(* Logix 5000 project; controller RG_Chopper vendor 1 type 14 code 235 rev 32.12; software revision 32.04; part 2 of 6 *)

ADD_ON_INSTRUCTION PUSH_PUSH_PB   (* revision 1.0, vendor JBT Food Tech *)
// Push Push (Dual State) Push Button
// Push - On; Push - Off
// Revision note:
// Rev 1.0 - 9/8/2010 - KM
VAR_INPUT
   HMI_PB : BOOL; {required}
   One_Shot : BOOL;
END_VAR
VAR_OUTPUT
   S_Out : BOOL; {access Read Only}
END_VAR
VAR_INPUT
   L_Out : BOOL; {visible}
END_VAR

ROUTINE Logic   (* ladder *)
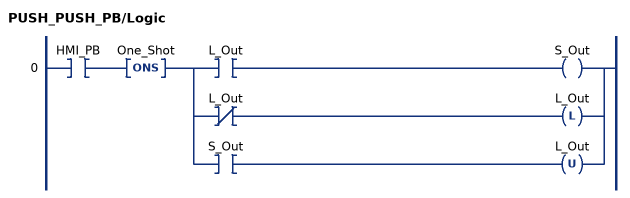
   0: XIC(HMI_PB)ONS(One_Shot)[XIC(L_Out) OTE(S_Out) ,XIO(L_Out) OTL(L_Out) ,XIC(S_Out) OTU(L_Out) ];
END_ROUTINE
END_ADD_ON_INSTRUCTION

ADD_ON_INSTRUCTION TD_TA_TP_4PORT_IOL   (* revision 1.0, vendor ifm efector *)
// Cyclic Data with Diagnostics
// Revision note:
// 4/27/17
VAR_IN_OUT
   PLC_Input : INT[123]; {required}
END_VAR
VAR_INPUT
   Port_Process_Data_Size : INT := 4; {visible}
   Port_Number : INT; {visible}
   Temp_Value_Gradient : REAL := 0.1; {visible}
END_VAR
VAR_OUTPUT
   Temperature : REAL; {access Read Only, visible}
   Vendor_ID : INT; {access Read Only, visible}
   Device_ID : INT; {access Read Only, visible}
   Datastorage_Error : BOOL; {access Read Only, visible}
   Process_Data : INT; {access Read Only}
   Device_Not_Connected : BOOL; {access Read Only, visible}
   IOL_Mode : BOOL; {access Read Only, visible}
   Invalid_Data : BOOL; {access Read Only, visible}
   Wrong_VID_DID : BOOL; {access Read Only, visible}
END_VAR
VAR
   RealPort_Num : INT; {access None}
   Offset_Address : INT; {access None}
   Process_PDI : INT; {access None}
   Process_Offset : INT; {access None}
   Offset_StatusFlgs : INT; {access None}
   StatusFlgs_Offset : INT; {access None}
   Data_Size : INT; {access None}
END_VAR

ROUTINE Logic   (* ladder *)
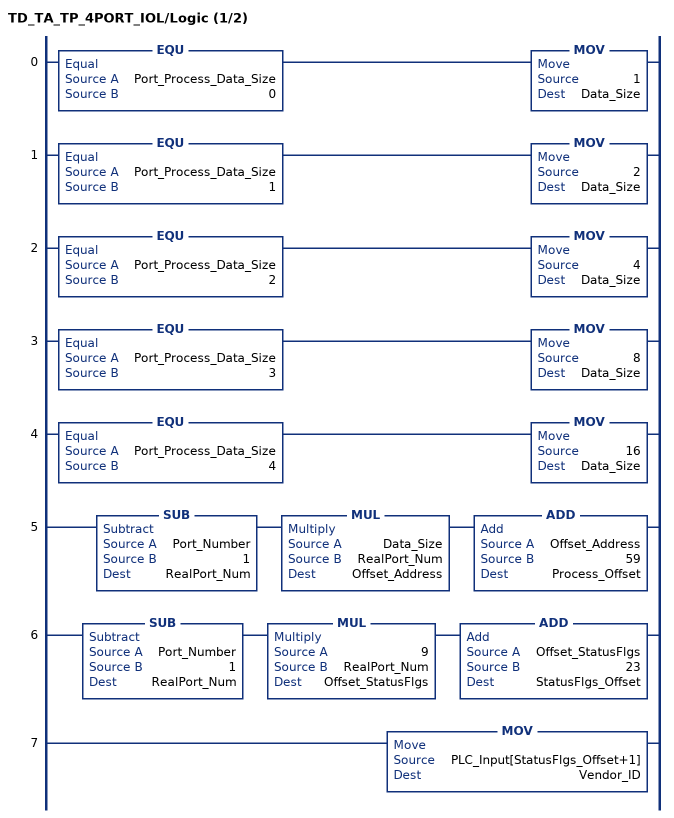
   0: EQU(Port_Process_Data_Size,0)MOV(1,Data_Size);
   1: EQU(Port_Process_Data_Size,1)MOV(2,Data_Size);
   2: EQU(Port_Process_Data_Size,2)MOV(4,Data_Size);
   3: EQU(Port_Process_Data_Size,3)MOV(8,Data_Size);
   4: EQU(Port_Process_Data_Size,4)MOV(16,Data_Size);
   5: SUB(Port_Number,1,RealPort_Num)MUL(Data_Size,RealPort_Num,Offset_Address)ADD(Offset_Address,59,Process_Offset);
   6: SUB(Port_Number,1,RealPort_Num)MUL(9,RealPort_Num,Offset_StatusFlgs)ADD(Offset_StatusFlgs,23,StatusFlgs_Offset);
   7: MOV(PLC_Input[StatusFlgs_Offset+1],Vendor_ID);
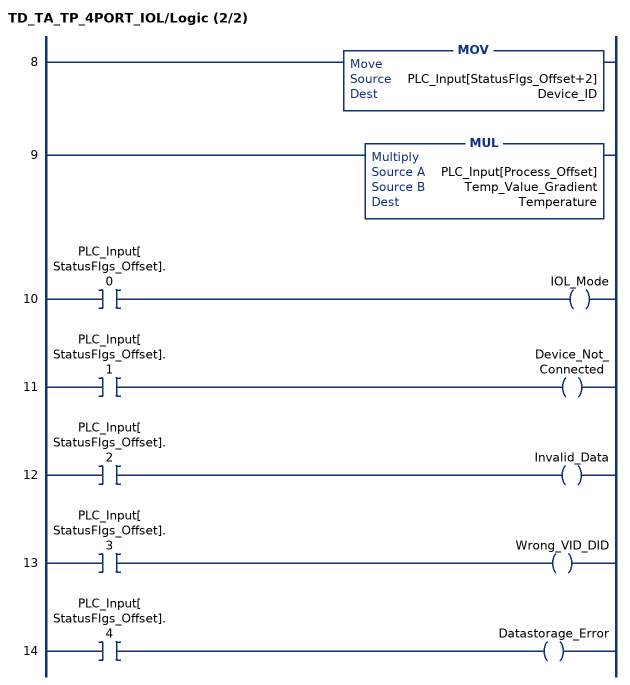
   8: MOV(PLC_Input[StatusFlgs_Offset+2],Device_ID);
   9: MUL(PLC_Input[Process_Offset],Temp_Value_Gradient,Temperature);
   10: XIC(PLC_Input[StatusFlgs_Offset].0)OTE(IOL_Mode);
   11: XIC(PLC_Input[StatusFlgs_Offset].1)OTE(Device_Not_Connected);
   12: XIC(PLC_Input[StatusFlgs_Offset].2)OTE(Invalid_Data);
   13: XIC(PLC_Input[StatusFlgs_Offset].3)OTE(Wrong_VID_DID);
   14: XIC(PLC_Input[StatusFlgs_Offset].4)OTE(Datastorage_Error);
END_ROUTINE
END_ADD_ON_INSTRUCTION

ADD_ON_INSTRUCTION TD_TA_TP_8PORT_IOL   (* revision 1.0, vendor ifm efector *)
// Cyclic Data with Diagnostics
// Revision note:
// 4/27/17
VAR_IN_OUT
   PLC_Input : INT[223]; {required}
END_VAR
VAR_INPUT
   Port_Process_Data_Size : INT := 4; {visible}
   Port_Number : INT; {visible}
   Temp_Value_Gradient : REAL := 0.1; {visible}
END_VAR
VAR_OUTPUT
   Temperature : REAL; {access Read Only, visible}
   Vendor_ID : INT; {access Read Only, visible}
   Device_ID : INT; {access Read Only, visible}
   Datastorage_Error : BOOL; {access Read Only, visible}
   Process_Data : INT; {access Read Only}
   Device_Not_Connected : BOOL; {access Read Only, visible}
   IOL_Mode : BOOL; {access Read Only, visible}
   Invalid_Data : BOOL; {access Read Only, visible}
   Wrong_VID_DID : BOOL; {access Read Only, visible}
END_VAR
VAR
   RealPort_Num : INT; {access None}
   Offset_Address : INT; {access None}
   Process_PDI : INT; {access None}
   Process_Offset : INT; {access None}
   Offset_StatusFlgs : INT; {access None}
   StatusFlgs_Offset : INT; {access None}
   Data_Size : INT; {access None}
END_VAR

ROUTINE Logic   (* ladder *)
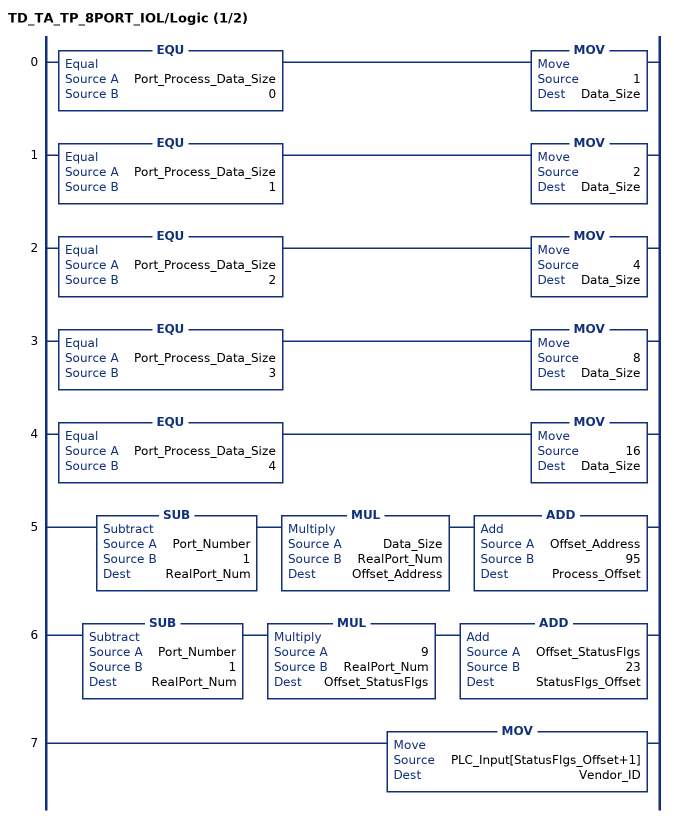
   0: EQU(Port_Process_Data_Size,0)MOV(1,Data_Size);
   1: EQU(Port_Process_Data_Size,1)MOV(2,Data_Size);
   2: EQU(Port_Process_Data_Size,2)MOV(4,Data_Size);
   3: EQU(Port_Process_Data_Size,3)MOV(8,Data_Size);
   4: EQU(Port_Process_Data_Size,4)MOV(16,Data_Size);
   5: SUB(Port_Number,1,RealPort_Num)MUL(Data_Size,RealPort_Num,Offset_Address)ADD(Offset_Address,95,Process_Offset);
   6: SUB(Port_Number,1,RealPort_Num)MUL(9,RealPort_Num,Offset_StatusFlgs)ADD(Offset_StatusFlgs,23,StatusFlgs_Offset);
   7: MOV(PLC_Input[StatusFlgs_Offset+1],Vendor_ID);
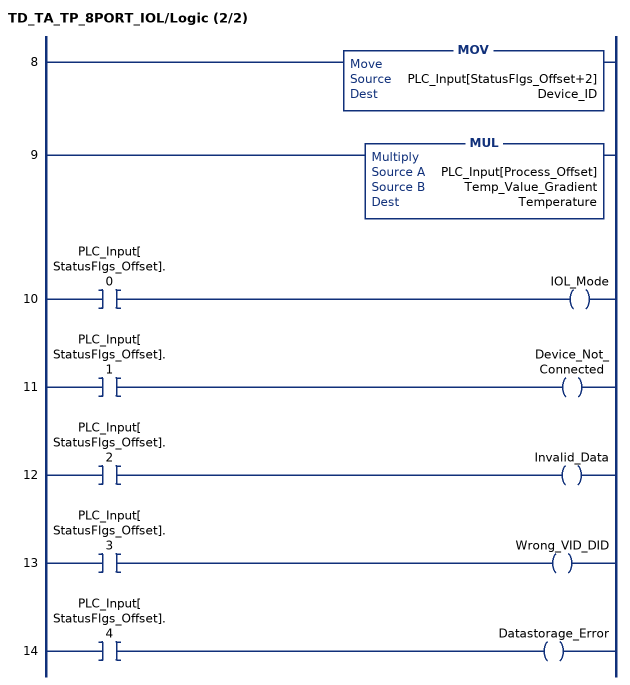
   8: MOV(PLC_Input[StatusFlgs_Offset+2],Device_ID);
   9: MUL(PLC_Input[Process_Offset],Temp_Value_Gradient,Temperature);
   10: XIC(PLC_Input[StatusFlgs_Offset].0)OTE(IOL_Mode);
   11: XIC(PLC_Input[StatusFlgs_Offset].1)OTE(Device_Not_Connected);
   12: XIC(PLC_Input[StatusFlgs_Offset].2)OTE(Invalid_Data);
   13: XIC(PLC_Input[StatusFlgs_Offset].3)OTE(Wrong_VID_DID);
   14: XIC(PLC_Input[StatusFlgs_Offset].4)OTE(Datastorage_Error);
END_ROUTINE
END_ADD_ON_INSTRUCTION

ADD_ON_INSTRUCTION TD_TA_TP_AL1020_IOL   (* revision 1.4, vendor ifm efector *)
// Cyclic Data with Diagnostics
// Revision note:
// Supports TDxxxx, TA2xxx, TP3xxx, TP9xxx
VAR_INPUT
   Port_Number : INT; {visible}
END_VAR
VAR_IN_OUT
   ioarybPLC_Input : INT[194]; {required}
END_VAR
VAR_OUTPUT
   Temp_Value : REAL; {access Read Only, required}
END_VAR
VAR_INPUT
   Temp_Value_Gradient : REAL := 0.1; {visible}
END_VAR
VAR_OUTPUT
   Vendor_ID : INT; {access Read Only, required}
   Device_ID : INT; {access Read Only, required}
   IOLinkmode_active : BOOL; {access Read Only, required}
   IOLink_communication : BOOL; {access Read Only, required}
   Device_Connected : BOOL; {access Read Only, required}
   Valid_Process_Data : BOOL; {access Read Only, required}
   Datastorage_error : BOOL; {access Read Only, required}
END_VAR
VAR
   ARYbInternInputData : INT[26]; {access None}
   Port1 : BOOL; {access None}
   Port2 : BOOL; {access None}
   Port3 : BOOL; {access None}
   Port4 : BOOL; {access None}
   Port5 : BOOL; {access None}
   Port6 : BOOL; {access None}
   Port7 : BOOL; {access None}
   Port8 : BOOL; {access None}
   Process_SWPB : INT; {access None}
END_VAR

ROUTINE Logic   (* ladder *)
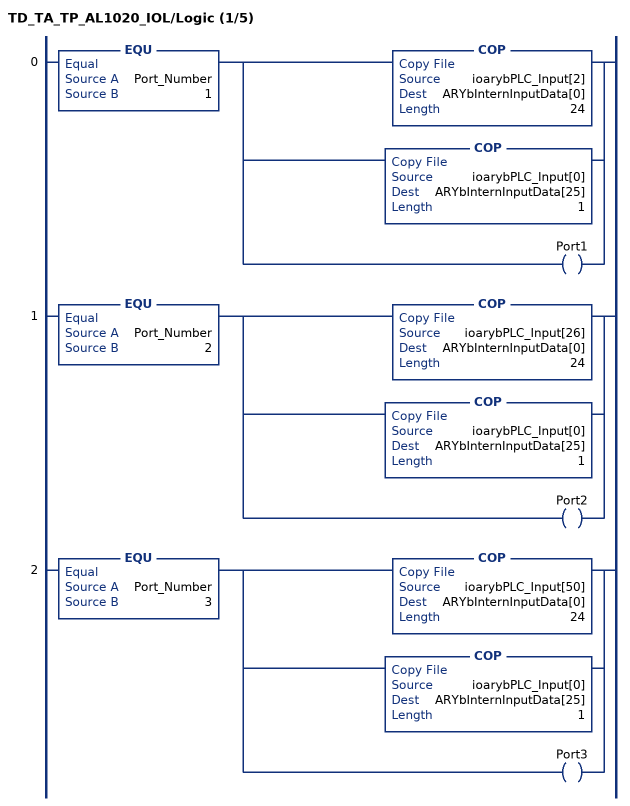
   0: EQU(Port_Number,1)[COP(ioarybPLC_Input[2],ARYbInternInputData[0],24) ,[COP(ioarybPLC_Input[0],ARYbInternInputData[25],1) ,OTE(Port1) ] ];
   1: EQU(Port_Number,2)[COP(ioarybPLC_Input[26],ARYbInternInputData[0],24) ,[COP(ioarybPLC_Input[0],ARYbInternInputData[25],1) ,OTE(Port2) ] ];
   2: EQU(Port_Number,3)[COP(ioarybPLC_Input[50],ARYbInternInputData[0],24) ,[COP(ioarybPLC_Input[0],ARYbInternInputData[25],1) ,OTE(Port3) ] ];
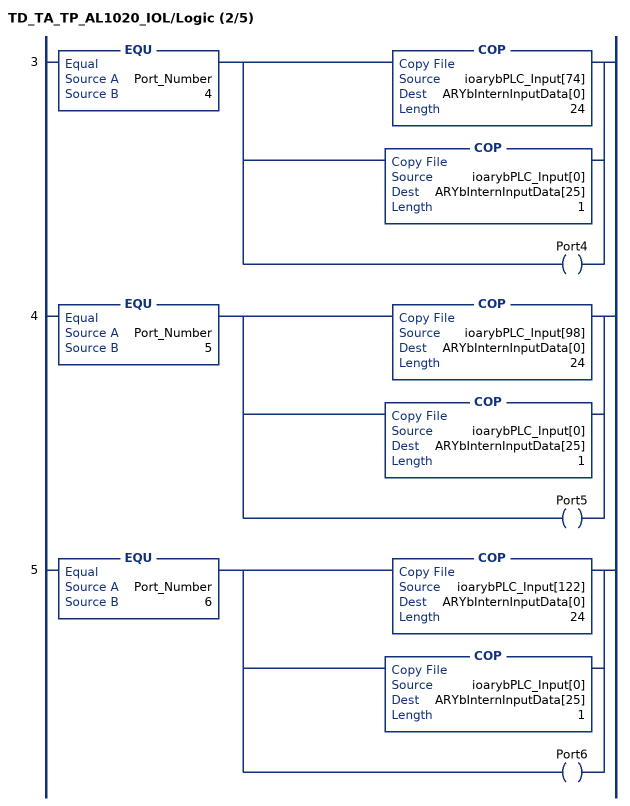
   3: EQU(Port_Number,4)[COP(ioarybPLC_Input[74],ARYbInternInputData[0],24) ,[COP(ioarybPLC_Input[0],ARYbInternInputData[25],1) ,OTE(Port4) ] ];
   4: EQU(Port_Number,5)[COP(ioarybPLC_Input[98],ARYbInternInputData[0],24) ,[COP(ioarybPLC_Input[0],ARYbInternInputData[25],1) ,OTE(Port5) ] ];
   5: EQU(Port_Number,6)[COP(ioarybPLC_Input[122],ARYbInternInputData[0],24) ,[COP(ioarybPLC_Input[0],ARYbInternInputData[25],1) ,OTE(Port6) ] ];
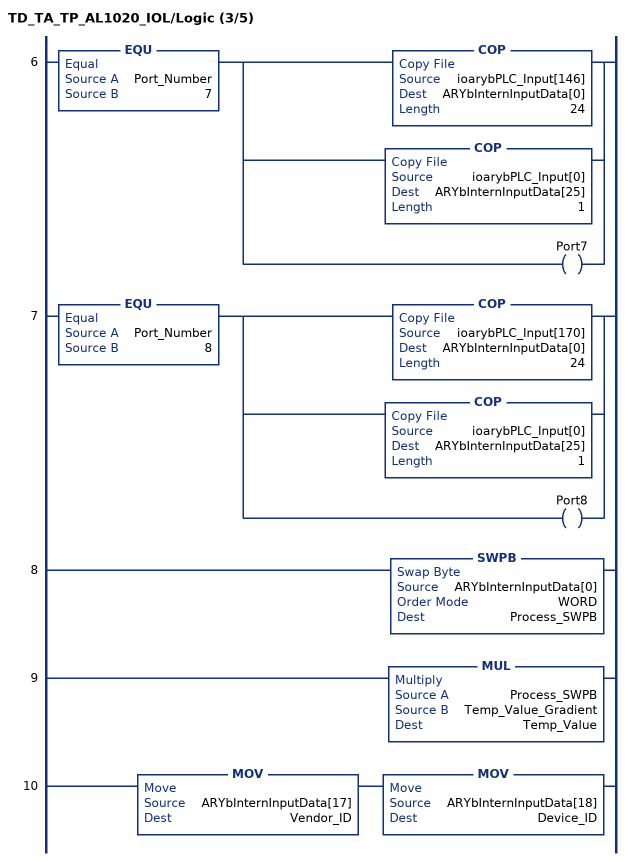
   6: EQU(Port_Number,7)[COP(ioarybPLC_Input[146],ARYbInternInputData[0],24) ,[COP(ioarybPLC_Input[0],ARYbInternInputData[25],1) ,OTE(Port7) ] ];
   7: EQU(Port_Number,8)[COP(ioarybPLC_Input[170],ARYbInternInputData[0],24) ,[COP(ioarybPLC_Input[0],ARYbInternInputData[25],1) ,OTE(Port8) ] ];
   8: SWPB(ARYbInternInputData[0],WORD,Process_SWPB);
   9: MUL(Process_SWPB,Temp_Value_Gradient,Temp_Value);
   10: MOV(ARYbInternInputData[17],Vendor_ID)MOV(ARYbInternInputData[18],Device_ID);
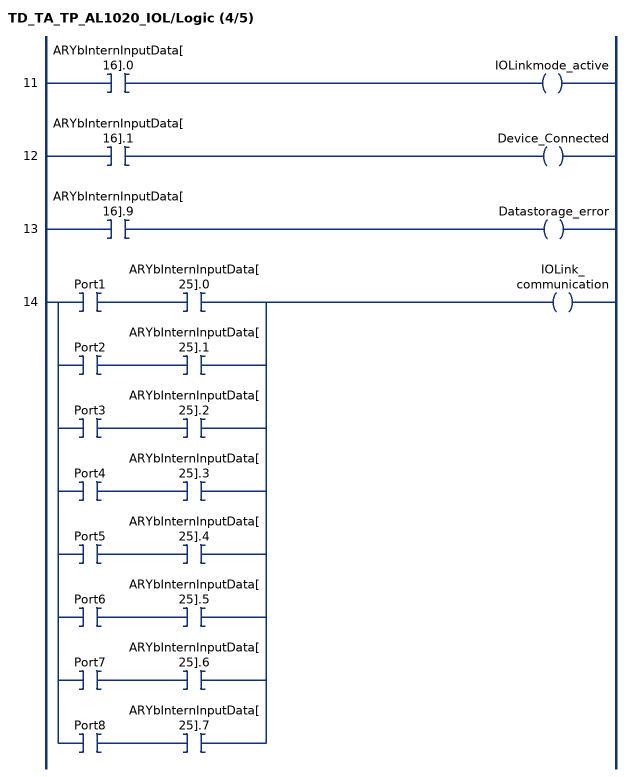
   11: XIC(ARYbInternInputData[16].0)OTE(IOLinkmode_active);
   12: XIC(ARYbInternInputData[16].1)OTE(Device_Connected);
   13: XIC(ARYbInternInputData[16].9)OTE(Datastorage_error);
   14: [XIC(Port1) XIC(ARYbInternInputData[25].0) ,[XIC(Port2) XIC(ARYbInternInputData[25].1) ,[XIC(Port3) XIC(ARYbInternInputData[25].2) ,[XIC(Port4) XIC(ARYbInternInputData[25].3) ,[XIC(Port5) XIC(ARYbInternInputData[25].4) ,[XIC(Port6) XIC(ARYbInternInputData[25].5) ,XIC(Port7) XIC(ARYbInternInputData[25].6) ,XIC(Port8) XIC(ARYbInternInputData[25].7) ] ] ] ] ] ]OTE(IOLink_communication);
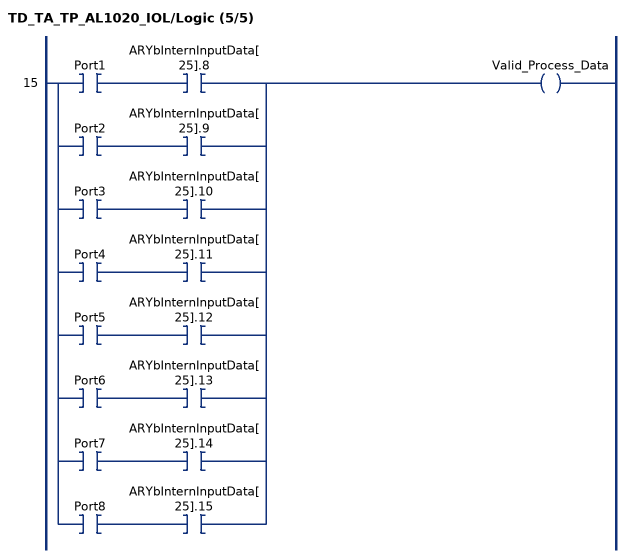
   15: [XIC(Port1) XIC(ARYbInternInputData[25].8) ,[XIC(Port2) XIC(ARYbInternInputData[25].9) ,[XIC(Port3) XIC(ARYbInternInputData[25].10) ,[XIC(Port4) XIC(ARYbInternInputData[25].11) ,[XIC(Port5) XIC(ARYbInternInputData[25].12) ,[XIC(Port6) XIC(ARYbInternInputData[25].13) ,XIC(Port7) XIC(ARYbInternInputData[25].14) ,XIC(Port8) XIC(ARYbInternInputData[25].15) ] ] ] ] ] ]OTE(Valid_Process_Data);
END_ROUTINE
END_ADD_ON_INSTRUCTION

ADD_ON_INSTRUCTION TK_CTRL   (* revision 1.0, vendor JBT Food Tech *)
// Tank Level Alarm / Control
// Revision note:
// Rev 1.0 - 9/7/2010 - KM
VAR_INPUT
   Anlg_In : REAL; {required}   // Raw Tank Level
END_VAR
VAR_OUTPUT
   Scaled_In : REAL; {required}   // Scaled Tank Level
END_VAR
VAR_INPUT
   Hi_SP_1 : REAL := 90.0; {visible}   // High Alarm 1 SP
   Hi_SP_2 : REAL := 50.0; {visible}   // High Alarm 2 SP
   Lo_SP_1 : REAL := 20.0; {visible}   // Low Alarm 1 SP
   Lo_SP_2 : REAL := 10.0; {visible}   // High Alarm 2 SP
END_VAR
VAR_OUTPUT
   Hi_AL_1 : BOOL; {visible}   // High Alarm 1 Output
   Hi_AL_2 : BOOL; {visible}   // High Alarm 2 Output
   Lo_AL_1 : BOOL; {visible}   // Low Alarm 1 Output
   Lo_AL_2 : BOOL; {visible}   // Low Alarm 2 Output
END_VAR
VAR_INPUT
   Alm_ACK_Hi1 : BOOL;   // High Alarm 1 ACK
   Alm_ACK_Hi2 : BOOL;   // High Alarm 2 ACK
   Alm_ACK_Lo1 : BOOL;   // Low Alarm 1 ACK
   Alm_ACK_Lo2 : BOOL;   // Low Alarm 2 ACK
   Alarm_ACK : BOOL;   // Global Alarm ACK
   Hi_INH_1 : BOOL; {visible}   // High Alarm 1 INHIBIT
   Hi_INH_2 : BOOL; {visible}   // High Alarm 2 INHIBIT
   Lo_INH_1 : BOOL; {visible}   // Low Alarm 1 INHIBIT
   Lo_INH_2 : BOOL; {visible}   // Low Alarm 2 INHIBIT
   A_RES_Hi1 : BOOL := 1; {visible}   // High Alarm 1 Automatic Reset EN
   A_RES_Hi2 : BOOL := 1; {visible}   // High Alarm 2 Automatic Reset EN
   A_RES_Lo1 : BOOL := 1; {visible}   // Low Alarm 1 Automatic Reset EN
   A_RES_Lo2 : BOOL := 1; {visible}   // Low Alarm 2 Automatic Reset EN
   R_Min : REAL; {visible}   // Scaling Raw Minimum
   R_Max : REAL := 1.0; {visible}   // Scaling Raw Maximum
   EU_Min : REAL; {visible}   // Scaling EU Minimum
   EU_Max : REAL := 1.0; {visible}   // Scaling EU Maximum
   Hi1_HIS : REAL := 10.0; {visible}   // High Alarm 1 Auto Reset Hysteresis
   Hi2_HIS : REAL := 10.0; {visible}   // High Alarm 2 Auto Reset Hysteresis
   Lo1_HIS : REAL := 10.0; {visible}   // Low Alarm 1 Auto Reset Hysteresis
   Lo2_HIS : REAL := 10.0; {visible}   // Low Alarm 2 Auto Reset Hysteresis
   Auto_RES_Hi1 : REAL;   // High Alarm 1 Calculated Reset Point
   Auto_RES_Hi2 : REAL;   // High Alarm 2 Calculated Reset Point
   Auto_RES_Lo1 : REAL;   // Low Alarm 1 Calculated Reset Point
   Auto_RES_Lo2 : REAL;   // Low Alarm 2 Calculated Reset Point
   Tmr1_PRE : REAL := 5.0; {visible}
   Tmr2_PRE : REAL := 5.0; {visible}
   Tmr3_PRE : REAL := 5.0; {visible}
   Tmr4_PRE : REAL := 5.0; {visible}
END_VAR
VAR
   Delay_4 : TIMER := (PRE := 5000); {access None}
   Delay_3 : TIMER := (PRE := 5000); {access None}
   Delay_2 : TIMER := (PRE := 5000); {access None}
   Delay_1 : TIMER := (PRE := 5000); {access None}
END_VAR

ROUTINE Logic   (* ladder *)
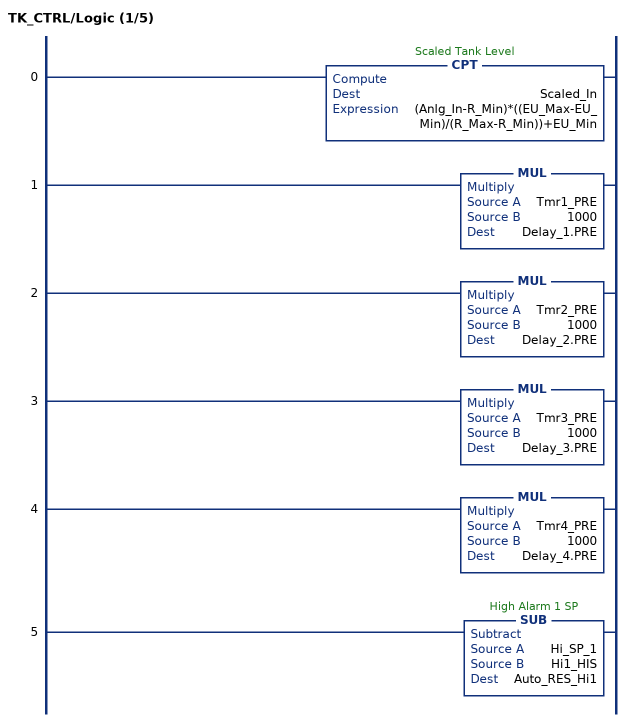
   0: CPT(Scaled_In,(Anlg_In-R_Min)*((EU_Max-EU_Min)/(R_Max-R_Min))+EU_Min);
   1: MUL(Tmr1_PRE,1000,Delay_1.PRE);
   2: MUL(Tmr2_PRE,1000,Delay_2.PRE);
   3: MUL(Tmr3_PRE,1000,Delay_3.PRE);
   4: MUL(Tmr4_PRE,1000,Delay_4.PRE);
   5: SUB(Hi_SP_1,Hi1_HIS,Auto_RES_Hi1);
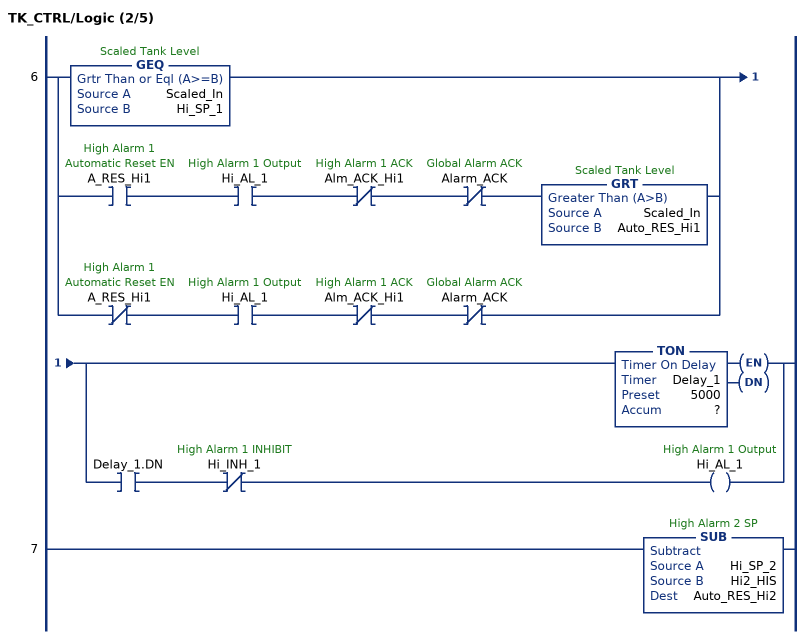
   6: [GEQ(Scaled_In,Hi_SP_1) ,XIC(A_RES_Hi1) XIC(Hi_AL_1) XIO(Alm_ACK_Hi1) XIO(Alarm_ACK) GRT(Scaled_In,Auto_RES_Hi1) ,XIO(A_RES_Hi1) XIC(Hi_AL_1) XIO(Alm_ACK_Hi1) XIO(Alarm_ACK) ][TON(Delay_1,?,?) ,XIC(Delay_1.DN) XIO(Hi_INH_1) OTE(Hi_AL_1) ];
   7: SUB(Hi_SP_2,Hi2_HIS,Auto_RES_Hi2);
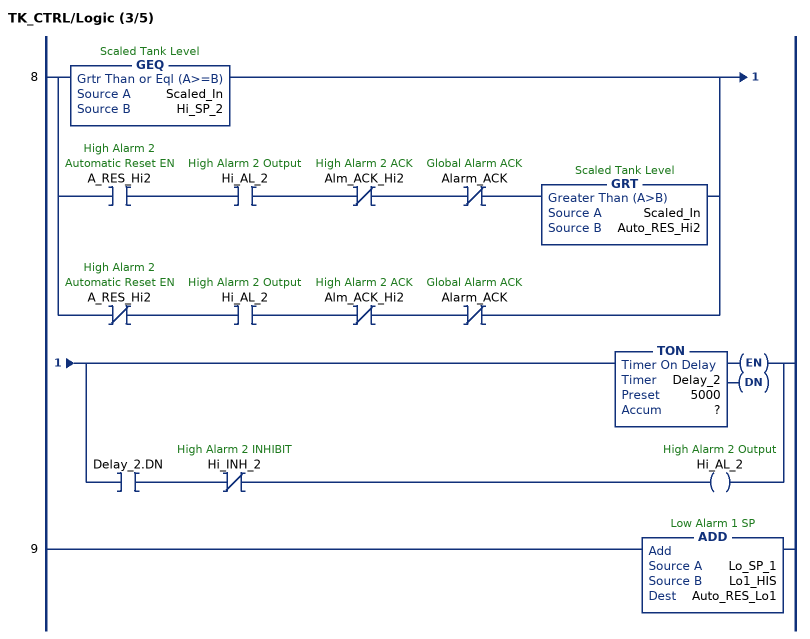
   8: [GEQ(Scaled_In,Hi_SP_2) ,XIC(A_RES_Hi2) XIC(Hi_AL_2) XIO(Alm_ACK_Hi2) XIO(Alarm_ACK) GRT(Scaled_In,Auto_RES_Hi2) ,XIO(A_RES_Hi2) XIC(Hi_AL_2) XIO(Alm_ACK_Hi2) XIO(Alarm_ACK) ][TON(Delay_2,?,?) ,XIC(Delay_2.DN) XIO(Hi_INH_2) OTE(Hi_AL_2) ];
   9: ADD(Lo_SP_1,Lo1_HIS,Auto_RES_Lo1);
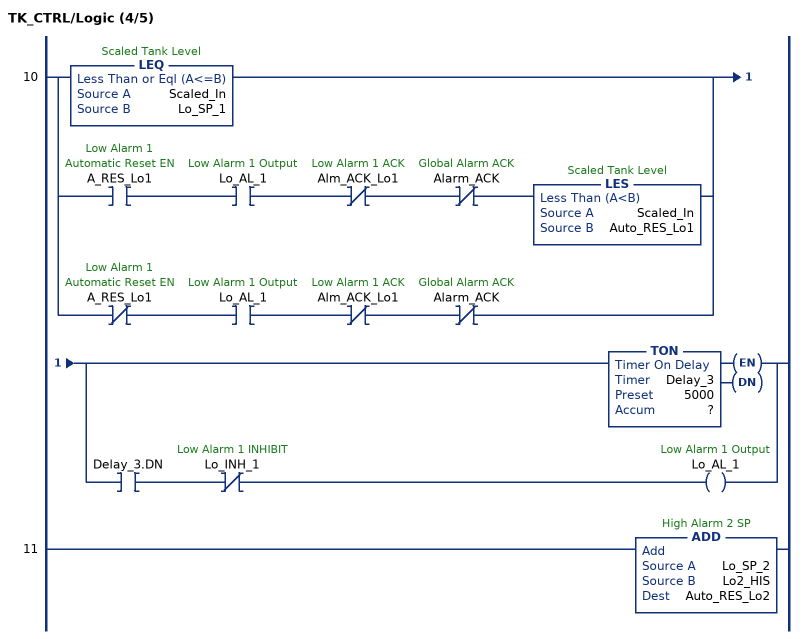
   10: [LEQ(Scaled_In,Lo_SP_1) ,XIC(A_RES_Lo1) XIC(Lo_AL_1) XIO(Alm_ACK_Lo1) XIO(Alarm_ACK) LES(Scaled_In,Auto_RES_Lo1) ,XIO(A_RES_Lo1) XIC(Lo_AL_1) XIO(Alm_ACK_Lo1) XIO(Alarm_ACK) ][TON(Delay_3,?,?) ,XIC(Delay_3.DN) XIO(Lo_INH_1) OTE(Lo_AL_1) ];
   11: ADD(Lo_SP_2,Lo2_HIS,Auto_RES_Lo2);
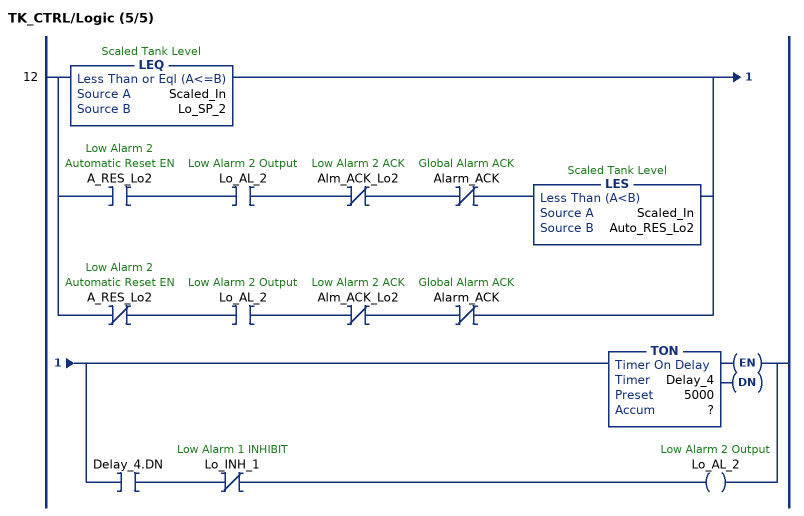
   12: [LEQ(Scaled_In,Lo_SP_2) ,XIC(A_RES_Lo2) XIC(Lo_AL_2) XIO(Alm_ACK_Lo2) XIO(Alarm_ACK) LES(Scaled_In,Auto_RES_Lo2) ,XIO(A_RES_Lo2) XIC(Lo_AL_2) XIO(Alm_ACK_Lo2) XIO(Alarm_ACK) ][TON(Delay_4,?,?) ,XIC(Delay_4.DN) XIO(Lo_INH_1) OTE(Lo_AL_2) ];
END_ROUTINE
END_ADD_ON_INSTRUCTION

ADD_ON_INSTRUCTION VLV_CTRL   (* revision 1.0, vendor JBT Food Tech *)
// Valve Control
// NO / NC
// No FeedBack
// Revision note:
// First Revision - 9/7/2010 - KM
VAR_INPUT
   AUTO_ALL : BOOL; {required}   // Global Device Auto
   Auto_PB : BOOL;   // - Auto Push Button
   Man_PB : BOOL;   // - Manual Push Button
   Off_PB : BOOL;   // - Off Push Button
END_VAR
VAR_OUTPUT
   Auto : BOOL; {visible}   // - Auto Status Output
   Man : BOOL; {visible}   // - Manual Status Output
   Off : BOOL; {visible}   // - Off Status Output
END_VAR
VAR_INPUT
   Vlv_DIS : BOOL;   // - Valve Disable
   _NC : BOOL; {required}   // Normally Closed Enable (For HMI Display)
   Auto_On : BOOL; {visible}   // - Automatic Output Control
END_VAR
VAR_OUTPUT
   Output : BOOL; {access Read Only, required}   // - Valve Output
   Vlv_St : BOOL; {access Read Only, visible}   // - Valve Status (On = Open)
END_VAR
VAR_INPUT
   Man_INH : BOOL; {access None, visible}   // - Manual Function Inhibit
   STOP : BOOL; {access None, required}   // - Global Stop
END_VAR

ROUTINE Logic   (* ladder *)
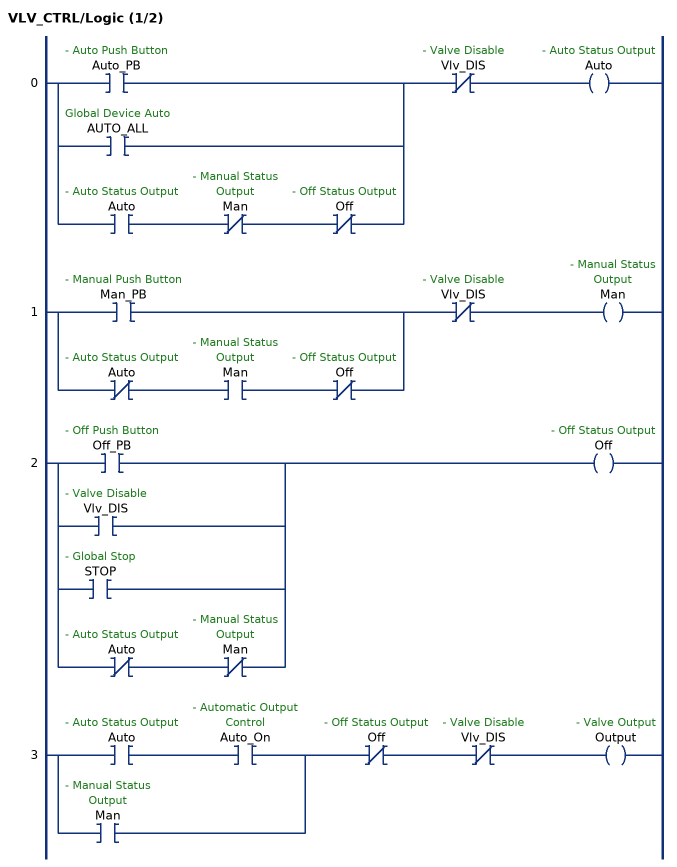
   0: [XIC(Auto_PB) ,XIC(AUTO_ALL) ,XIC(Auto) XIO(Man) XIO(Off) ]XIO(Vlv_DIS)OTE(Auto);
   1: [XIC(Man_PB) ,XIO(Auto) XIC(Man) XIO(Off) ]XIO(Vlv_DIS)OTE(Man);
   2: [XIC(Off_PB) ,XIC(Vlv_DIS) ,XIC(STOP) ,XIO(Auto) XIO(Man) ]OTE(Off);
   3: [XIC(Auto) XIC(Auto_On) ,XIC(Man) ]XIO(Off)XIO(Vlv_DIS)OTE(Output);
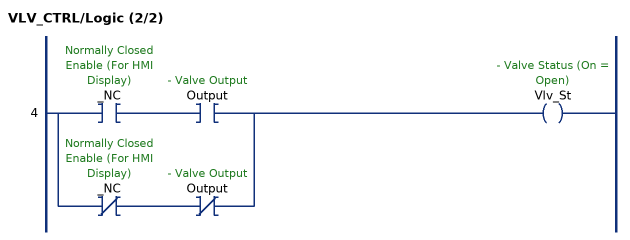
   4: [XIC(_NC) XIC(Output) ,XIO(_NC) XIO(Output) ]OTE(Vlv_St);
END_ROUTINE
END_ADD_ON_INSTRUCTION

VAR_GLOBAL   (* controller tags *)
   _CB103_VSD_AUX : BOOL;   // Local:1:I.Data.10
   _DBL101_TANK_LEVEL : BOOL;   // Conentrate Chopper Level Switch Local:1:I.Data.9
   _DBS101_DUMPER_SR : BOOL;   // Local:1:I.Data.11
   _ILG101_GREEN_PB : BOOL := 1;   // Green Light Pushbutton Local:1:O.Data.2
   Ack_All : BOOL;
   ALARM_FATAL : BOOL;   // Fatal Alarm Stops All Operation
   ALARM_GATE_OPEN : BOOL;   // Gate Open
   ALARM_LIGHT_CUR : BOOL;   // Light Curtain Obstructed
   ALARM_NON_FATAL : BOOL;
   Alarm_Reset_1 : BOOL;
   ALARM_S_FATAL : BOOL;   // Fatal Alarm Safety Map Stops All Operation
   ALARM_S_NON_FATAL : BOOL;   // Alarm Non-Fatal Safety Map
   AUTO_ALL : BOOL;   // All Devices to AUTO
   BLANK_LVL_DISP : BOOL := 1;   // Disables Tank Level Display
   CB104_DUMPER_AUX : BOOL := 1;   // CB104 Dumper Aux From Dumper Control
   CIP_CAUSTIC_RUNNING : ALIAS FOR SIGNAL_OUT_RG_CHOPPER.4;
   CIP_CMPLT : BOOL;   // CIP Complete Indicator
   CIP_COMPLETE : ALIAS FOR SIGNAL_IN_RG_CHOPPER.4;
   CIP_CYC_ST : DINT;   // CIP Cycle Status HMI
   CIP_OUT : DINT;   // CIP Output Bits
   CIP_REQUEST : ALIAS FOR SIGNAL_OUT_RG_CHOPPER.2;
   CIP_STEP : COUNTER := (PRE := 8);   // CIP Step Counter
   CIP_STEP_BIT : DINT;   // CIP Step Enable Bit
   CIP_STEP_DN : BOOL;   // CIP Step Done
   CIP_STEP_TMR : TIMER := (PRE := 900000);   // CIP Step Timer
   CIP_STP_TM_TB : DINT[13] := ([0] := 1000, [1] := 5000, [2] := 900000, [3] := 5000, [4] := 1800000, [5] := 5000, [6] := 28800000, [7] := 5000, [8] := 15000, [9] := 1000, [10] := 1000, [11] := 1000, [12] := 1000); {constant}   // CIP Step Timer PreSet Table
        [0]   // CIP Step Timer PreSet Step #0
        [10]   // CIP Step Timer PreSet Step #10
        [11]   // CIP Step Timer PreSet Step #11
        [12]   // CIP Step Timer PreSet Step #12
        [1]   // CIP Step Timer PreSet Step #1
        [2]   // CIP Step Timer PreSet Step #2
        [3]   // CIP Step Timer PreSet Step #3
        [4]   // CIP Step Timer PreSet Step #4
        [5]   // CIP Step Timer PreSet Step #5
        [6]   // CIP Step Timer PreSet Step #6
        [7]   // CIP Step Timer PreSet Step #7
        [8]   // CIP Step Timer PreSet Step #8
        [9]   // CIP Step Timer PreSet Step #9
   CIP_STRT_RUN : BOOL;   // CIP System Started
   CIP_WATER_RUNNING : ALIAS FOR SIGNAL_OUT_RG_CHOPPER.3;
   CYC_CIP : BOOL;   // CIP Cycle Running
   CYC_RUN : BOOL := 1;   // Production Cycle Running
   CYC_ST : DINT := 1;
   DBT101 : TD_TA_TP_8PORT_IOL := (Port_Process_Data_Size := 4, Port_Number := 2, Temp_Value_Gradient := 0.1, Temperature := 11.3, Vendor_ID := 310, Device_ID := 140, IOL_Mode := 1);   // DTT101 Hot Water Temperature IO-Link RAW
   DBT101_RAW : REAL;   // DTT101 Hot Water Temperature
   DBT102 : TD_TA_TP_8PORT_IOL := (Port_Process_Data_Size := 4, Port_Number := 3, Temp_Value_Gradient := 0.1, Temperature := 9.1, Vendor_ID := 310, Device_ID := 141, IOL_Mode := 1);   // DBT102 Product Temperature IO-Link RAW
   DBX101_AM : PUSH_PUSH_PB;   // DBX-101 Push-Push Button Control
   DBX101_AUX : BOOL;   // DBX-101 Agitator Motor Aux
   DBX101_CTL : HOA_CTRL_v2 := (Off := 1, Auto_Run := 1, FB_EN := 1);   // DBX-101 Agitator Motor Control Block
   DBX101_CTL_ST : DINT := 2;   // DBX-101 Control Status 0= Auto 1= Manual 2= Error
   DBX101_FAULT : BOOL;
   DBX101_MAN : PUSH_PUSH_PB;   // DBX-101 Manual Run Push-Push
   DBX101_MAN_RUN : BOOL;   // DBX-101 Manual Run
   DBX101_MAN_ST : DINT := 2;   // DBX-101 Manual Control Status
   DBX101_OL : BOOL;   // DBX-101 Motor OverLoad Status
   DBX101_OUT : BOOL;   // DBX-101 Control Output
   DBX101_PB : BOOL;   // DBX-101 Auto / Manual Push-Push Button
   DBX101_S_START : BOOL;   // DBX-101 Safety map Agitator Start
   DBX101_START : BOOL;   // DBX-101 Agitator Start Safety Mapped DBX101_S_START
   DBX101_STS : DINT;   // DBX-101 Agitator Motor Status (HMI)
   DBX102_AM : PUSH_PUSH_PB;   // DBX-102 Push-Push Button Control
   DBX102_AUX : ALIAS FOR SIGNAL_IN_RG_CHOPPER.0;   // DBX-102 VFD Active AUX
   DBX102_CTL : HOA_CTRL_v2 := (Off := 1, Auto_Run := 1);   // DBX102 Product Discharge Pump Control Block
   DBX102_CTL_ST : DINT := 1;   // DBX-102 Control Status 0= Auto 1= Manual 2= Error
   DBX102_EN : BOOL := 1;   // DBX-102 VFD Safety ENABLE
   DBX102_ENABLE : ALIAS FOR SIGNAL_IN_RG_CHOPPER.1;
   DBX102_FAULT : BOOL;   // DBX-102 Discharge Pump Drive Fault
   DBX102_M_FAULT : BOOL;   // DBX-102 Discharge Pump Drive or Motor Fault
   DBX102_MAN : PUSH_PUSH_PB;   // DBX-102 Manual Control Push-Push
   DBX102_MAN_RUN : BOOL;   // DBX-102 Manual Mode Run PB
   DBX102_MAN_ST : DINT := 2;   // DBX-102 Manual Control Status
   DBX102_OUT : BOOL;   // DBX-102 Intermidiate Motor Control Output
   DBX102_PB : BOOL;   // DBX-102 Auto / Manual Push-Push Button
   DBX102_SPD : ANLG_SCALE := (Anlg_In := 100.0, RAW_Max := 100.0, EU_Max := 6000.0, Anlg_Scaled := 6000.0);   // DBX-102 Product Pump Speed Scaling
   DBX102_SPD_AM : PUSH_PUSH_PB := (L_Out := 1);   // DBX-102 Speed Push-Push Button Control
   DBX102_SPD_IN : REAL := 100.0;   // DBX-102 Product Pump User Requested Speed
   DBX102_SPD_OUT : REAL;   // DBX-102 VFD Alternate Requested Speed
   DBX102_SPD_PB : BOOL;   // DBX-102 Speed Auto / Manual PB
   DBX102_SPD_REQ : REAL := 100.0;   // DBX-102 VFD Requested Speed
   DBX102_SPD_ST : DINT := 1;   // DBX-102 VFD Speed Control Status 0= Auto 1= Manual 2= Error
   DBX102_START : BOOL;   // DBX-102 Product Pump VFD START
   DBX102_STS : DINT;   // DBX-102 Product Pump Status (HMI)
   DBX102_VFD_FB : ANLG_SCALE := (RAW_Max := 6000.0, EU_Max := 100.0);   // DBX-102 VFD Speed FB Scaling (HMI)
   DBX102_VFD_FB_SCL : REAL;   // DBX-102 Product Pump VFD Speed FB Scaling (HMI)
   DBX102B_EN : BOOL;   // DBX-102 Drive Enable
   DBX102B_S_En : BOOL := 1;   // DBX-102 Drive Safety Enable
   DBX103_AM : PUSH_PUSH_PB;   // DBX-103 Push-Push Button Control
   DBX103_AUX : BOOL;   // DBX-103 Water Pump Aux
   DBX103_CTL : HOA_CTRL_v2 := (Off := 1, Auto_Run := 1);   // DBX-103 Hot Water Pump Control Block
   DBX103_CTL_ST : DINT := 2;   // DBX-103 Control Status 1= Auto 2= Manual 3= Error
   DBX103_FAULT : BOOL;   // DBX-103 Hot Water Pump Fault
   DBX103_MAN : PUSH_PUSH_PB;   // DBX-103 Manual Run Push-Push
   DBX103_MAN_RUN : BOOL;   // DBX-101 Manual Run
   DBX103_MAN_ST : DINT := 2;   // DBX-103 Manual Control Status
   DBX103_OL : BOOL;   // DBX-103 Motor OverLoad Status
   DBX103_OUT : BOOL;   // DBX-103 Control Output
   DBX103_PB : BOOL;   // DBX-103 Auto / Manual Push-Push Button
   DBX103_S_START : BOOL;   // DBX-103 Safety map Hot Water Pump Start
   DBX103_START : BOOL;   // DBX-103 Water Pump Start Safety Mapped DBX103_S_START
   DBX103_STS : DINT;   // DBX-103 Hot Water Pump Status (HMI)
   DBX104_AM : PUSH_PUSH_PB := (L_Out := 1);   // DBX-104 Push-Push Button Control
   DBX104_AUX : BOOL;   // DBX-104 VFD Active AUX
   DBX104_CTL : HOA_CTRL_v2 := (Off := 1, Man_INH := 1, TB_AM := 1);   // DBX-104 Reversing Motor Starter Control
   DBX104_CTL_ST : DINT := 2;   // DBX-104 Control Status 0= Auto 1= Manual 2= Error
   DBX104_DD : PUSH_PUSH_PB;   // DBX104 VFD Direction DOWN Control
   DBX104_DIRCT : BOOL;   // DBX-104 Drum Dumper VFD Direction 0 = DOWN 1 = UP
   DBX104_DU : PUSH_PUSH_PB;   // DBX104 VFD Direction UP Control
   DBX104_DWN : BOOL;   // DBX-104 Drum Dumper VFD Direction DOWN
   DBX104_EN : BOOL;   // DBX-104 Brake Safety ENABLE
   DBX104_FAULT : BOOL;   // DBX-104 Dumper Elevator Drive Fault
   DBX104_M_FAULT : BOOL;   // DBX-104 Dumper Elevator Drive or Motor Fault
   DBX104_MAN : PUSH_PUSH_PB := (One_Shot := 1);   // DBX-104 Manual Control Push-Push
   DBX104_MAN_RUN : BOOL;   // DBX-104 Manual Mode Run PB
   DBX104_MAN_ST : DINT := 2;   // DBX-104 Manual Control Status
   DBX104_PB : BOOL;   // DBX-104 Auto / Manual Push-Push Button
   DBX104_S_DIR_EN : BOOL := 1;   // DBX-104 Dump Elevator Direction Enabled
   DBX104_S_DWN : BOOL;   // DBX-104 Dump Elevator DOWN (Safety)
   DBX104_S_START : BOOL;   // DBX-104 Dump Elevator START (Safety)
   DBX104_S_UP : BOOL;   // DBX-104 Dump Elevator UP (Safety)
   DBX104_SPD : ANLG_SCALE := (Anlg_In := 100.0, RAW_Max := 100.0, EU_Max := 6000.0, Anlg_Scaled := 6000.0);   // DBX-104 Product Pump Speed Scaling
   DBX104_SPD_AM : PUSH_PUSH_PB;   // DBX-104 Speed Push-Push Button Control
   DBX104_SPD_IN : DINT := 100;   // DBX-102 Product Pump User Requested Speed
   DBX104_SPD_OUT : DINT;   // DBX-104 VFD Alternate Requested Speed
   DBX104_SPD_PB : BOOL;   // DBX-104 Speed Auto / Manual PB
   DBX104_SPD_REQ : DINT := 100;   // DBX-104 VFD Requested Speed
   DBX104_SPD_ST : DINT;   // DBX-104 VFD Speed Control Status 0= Auto 1= Manual 2= Error
   DBX104_START : BOOL;   // DBX-104 Drum Dumper VFD START
   DBX104_STS : DINT;   // DBX-104 Product Pump Status (HMI)
   DBX104_UP : BOOL;   // DBX-104 Drum Dumper VFD Direction UP
   DBX104_VFD_FB : ANLG_SCALE := (RAW_Max := 6000.0, EU_Max := 100.0);   // DBX-104 VFD Speed FB Scaling (HMI)
   DBX104_VFD_FB_SCL : REAL;   // DBX-104 Product Pump VFD Speed FB Scaling (HMI)
   DBX104B_EN : BOOL;   // DBX-104 Brake Enable
   DBX104B_S_En : BOOL := 1;   // DBX-104 Drive Enable Safety
   deleteme : DINT;
   deletemeS : BOOL;
   DL101_In : REAL;
   DL101_Scl : REAL := 0.9174312;
   DLT101 : PN_PI_PP_8PORT_IOL := (Port_Process_Data_Size := 4, Port_Number := 1, IOL_Mode := 1, Pressure_Gradient := 0.1, Pressure := 1.0, Vendor_ID := 310, Device_ID := 257, Out2 := 1);   // DLT101 Tank Level IO-Link RAW
   DLT101_LVL_SCL : REAL := 0.9174312;   // Tank Level Scaled (0.0 - 100.0%)
   DLT101_SCL : ANLG_SCALE := (Anlg_In := 1.0, RAW_Min := 0.5, RAW_Max := 55.0, EU_Max := 100.0, Anlg_Scaled := 0.9174312);   // Tank Level Scaling Block
   DLT101_Tk : TK_CTRL := (Anlg_In := 0.9174312, Scaled_In := 0.9174312, Hi_SP_1 := 90.0, Hi_SP_2 := 50.0, Lo_SP_1 := 20.0, Lo_SP_2 := 5.0, Lo_AL_1 := 1, Lo_AL_2 := 1, A_RES_Hi1 := 1, A_RES_Hi2 := 1, A_RES_Lo1 := 1, A_RES_Lo2 := 1, R_Max := 100.0, EU_Max := 100.0, Hi1_HIS := 10.0, Hi2_HIS := 10.0, Lo1_HIS := 10.0, Lo2_HIS := 5.0, Auto_RES_Hi1 := 80.0, Auto_RES_Hi2 := 40.0, Auto_RES_Lo1 := 30.0, Auto_RES_Lo2 := 10.0, Tmr1_PRE := 5.0, Tmr2_PRE := 5.0, Tmr3_PRE := 5.0, Tmr4_PRE := 5.0);   // Tank Level Control
   DTT101 : REAL := 52.34;   // DTT-101 Hot Water Temperature Analong In
   DTT102 : REAL := 48.38;   // Discharge Product Temperature
   Dual_Mon_1 : DCI_MONITOR;
   Dual_Mon_2 : DCI_MONITOR;
   Dual_Mon_3 : DCI_MONITOR;
   DWN_MKBK : BOOL;   // Elevator Down Make / Break LS_L1 Detection
   DWN_MKBK1 : BOOL := 1;   // Elevator Down Make / Break Memory 1
   DWN_OT_AL : BOOL;   // New Dumper DOWN Over Travel Alarm
   DWN_STP : BOOL := 1;   // Elevator Down STOP
   Fault_ACK : BOOL;   // Fault Acknowledge
   FAULT_ACK_PB : BOOL;   // Fault ACK Push Button
   FAULT_NOTIFICATION : ALIAS FOR SIGNAL_OUT_RG_CHOPPER.12;
   Flash : BOOL;
   Flash_S : BOOL;   // Safety Flash Bit
   Gate_SW1 : DCI_MONITOR := (ChannelA := 1, ChannelB := 1, InputStatus := 1, SafetyFunction := 41, DiscrepancyTime := 200, O1 := 1, IS := 1);   // Safety Switch Gate_SW1 SW105 A/B
   Gate_SW2 : DCI_MONITOR := (ChannelA := 1, ChannelB := 1, InputStatus := 1, SafetyFunction := 41, DiscrepancyTime := 200, O1 := 1, IS := 1);   // Safety Switch Gate_SW2 SW108 A/B
   HI_PROD_TEMP_AL : BOOL;   // Product Temperature High Alarm
   HI_PROD_TEMP_SP : REAL;   // Product High Temperature Alarm SetPoint
   HI_TMP_TMR : TIMER := (PRE := 10000);   // Product Temperature High Alarm Timer
   HMI_FLT_RES : BOOL;   // Safety Module Fault Reset HMI
   HMI_USER : STRING;   // Current Logged HMI User
   HT_TEMP_SP : REAL := 105.0;   // TCV-101 SetPoint from HMI
   ILG104_GREEN_STACK : BOOL := 1;   // Stack Light Green
   ILG105_YELLOW_STACK : BOOL;   // Stack Light Yellow
   ILG106_RED_STACK : BOOL;   // Stack Light Red
   ILR102_RED_PB : BOOL;   // Red Light Pushbutton
   INTERLOCK_TMR1 : TIMER := (PRE := 25, EN := 1, DN := 1);   // DBX-104 Safety Interlock Timer
   INTERLOCK_TMR2 : TIMER := (PRE := 25, EN := 1, DN := 1);   // DBX-102 Safety Interlock Timer
   KR101_DUMPER_PERM : BOOL := 1;   // Dumper Permissive NON-FATAL ALARM 0 = ALARM
   L_CRASH_ALM : BOOL;   // New Dumper Lower CRASH Alarm
   LEVEL_TIMER : TIMER := (PRE := 120000);   // Juice Tank At High Level
   LOT1_TMR : TIMER := (PRE := 2000, ACC := 2000);   // Lower Over Travel Switch Disable Timer
   LS_L1 : BOOL := 1;   // New Dumper LOWER Limit Switch #1
   LS_LID_OPN : BOOL := 1;   // Lid Open Switch IO-Link Master Mapped X04
   LS_M1 : BOOL;   // New Dumper MIDDLE Limit Switch #1
   LS_U1 : BOOL;   // New Dumper UPPER Limit Switch #1
   LSS_L2 : BOOL := 1;   // New Dumper LOWER Safety Limit Switch #2
   LSS_LOT1 : BOOL;   // New Dumper LOWER OVER TRAVEL Limit Switch
   LSS_U2 : BOOL;   // New Dumper UPPER Safety Limit Switch #2
   LVL_BLANK_SP : REAL := 4.0;   // Real Value Below Blanks Level Display
   LVL_LO_TMR : TIMER := (PRE := 2000, ACC := 2000, EN := 1, DN := 1);   // Low Tank Level Alarm Debounce Timer
   M104S_DWN_CTL : CONFIGURABLE_ROUT := (Feedback1 := 1, Feedback2 := 1, InputStatus := 1, OutputStatus := 1, FeedbackReactionTime := 500);   // DBX-104 Dump Elevator Safety Starter Down Output
   M104S_STRT_CTL : CONFIGURABLE_ROUT := (Feedback1 := 1, Feedback2 := 1, InputStatus := 1, OutputStatus := 1, FeedbackReactionTime := 500);   // DBX-104 Dump Elevator Safety Starter Enable Output
   M104S_UP_CTL : CONFIGURABLE_ROUT := (Feedback1 := 1, Feedback2 := 1, InputStatus := 1, OutputStatus := 1, FeedbackReactionTime := 500);   // DBX-104 Dump Elevator Safety Starter UP Output
   NO_USER : BOOL := 1;   // No HMI User Logged on
   ONESHOT : DINT := 537373125;   // One-shot Word
   PB101 : BOOL;   // Drum Dumper Elevator UP Push Button
   PB102 : BOOL;   // Drum Dumper Elevator DOWN Push Button
   PB103 : BOOL;   // Drum Dumper Elevator STOP Push Button
   PCV101_AO_SCL : REAL;   // PCV-101 Hot Water Temperature Control Scaled Output
   PCV101_SCL : ANLG_SCALE := (RAW_Max := 100.0, EU_Max := 100.0);   // PCV-101 Temperature Control Scaling Block
   PROC_TMR : TIMER[16] := ([1].PRE := 5000, [1].ACC := 5000, [1].EN := 1, [1].DN := 1, [2].PRE := 5000, [2].ACC := 5000, [2].EN := 1, [2].DN := 1, [3].PRE := 10000, [6].PRE := 3000, [7].PRE := 3000, [8].PRE := 3000, [9].PRE := 5000, [10].PRE := 10000, [11].PRE := 29000);   // Process Timers
   S_ESTOP : BOOL := 1;   // Safety ESTOP
   S_ESTOP_1 : EMERGENCY_STOP := (ResetType := 1, ChannelA := 1, ChannelB := 1, O1 := 1);   // Safety ESTOP Block #1
   S_ESTOP_2 : EMERGENCY_STOP := (ResetType := 1, ChannelA := 1, ChannelB := 1, O1 := 1);   // Safety ESTOP Block #2
   S_Fault_Res : BOOL;   // Safety Circuit Fault Reset
   S_HORN : BOOL;   // Audible Alarm HORN
   S_SW_IN : DINT := 29375547;   // Safety Switch Input Array
        .0   // E-Stop Main ESTOP_1A
        .1   // E-Stop Main ESTOP_1B
        .10   // Safety Switch Dumper Light Curtain SW106A
        .11   // Safety Switch Dumper Light Curtain SW106B
        .12   // Safety Switch Gate Switch #2 SW108A
        .13   // Safety Switch Gate Switch #2 SW108B
        .17   // Module Fault RESET
        .2   // Safety Trip RESET PB PB2361
        .22   // M104 Elevator Motor Starter AUX (Safety)
        .23   // M104 Elevator Motor Start Forward AUX (Safety)
        .24   // M104 Elevator Motor Start Reverse AUX (Safety)
        .3   // E-Stop Dumper ESTOP_2 SCR-1291
        .4   // Safety Switch Gate SW #1 SW105A
        .5   // Safety Switch Gate SW #1 SW105B
        .6   // Safety Switch Tank Lid SW107A
        .7   // Safety Switch Tank Lid SW107B
        .8   // Safety Switch Gate SW #2 SW108A
   S_SW_OUT : DINT;   // Safety Switch Output Array
   S_TEST : DINT := 1;   // Safety Test Bits
   S_TMR_1 : TIMER := (PRE := 1000, ACC := 640, EN := 1, TT := 1);   // Safety Timer #1
   S_TMR_2 : TIMER := (PRE := 1000);   // Safety Timer #2
   SCR1291 : BOOL := 1;   // Dumper Estop Permissive Lost SCR-1291
   SCRL_STRT : TIMER := (PRE := 500);   // Scroll Startup Warning Timer
   SHTDWN_ACTV : BOOL;   // System Shutdown is In Progress
   SHTDWN_CMPLT : BOOL;   // System Shutdown Complete
   SHUTDOWN : DINT;   // System Shutdown Control Bits
        .6   // System Shutdown Time-out
   SIGNAL_IN_RG_CHOPPER : DINT := 2;
        .0   // Remote Signal Input DBX-102 Running
        .1   // Remote Signal Input DBX-102 Enable
        .2   // Remote Signal Input Water Running
        .3   // Remote Signal Input Caustic Running
        .4   // Remote Signal Input CIP Complete
   SIGNAL_OUT_RG_CHOPPER : DINT := 9730;
        .0   // Remote Signal Output DBX-102 Start
        .1   // Remote Signal Output Steam Enable
        .10   // Remote Signal Output SW-104 ESTOP
        .11   // Remote Signal Output CIP Complete
        .12   // Remote Signal Output CIP FAULT
        .13   // Remote Signal Output SW-108 ESTOP 2
        .2   // Remote Signal Output CIP Request / Enable
        .3   // Remote Signal Output CIP Water Request
        .4   // Remote Signal Output CIP Caustic Request
        .5   // Remote Signal Output SW-105 Gate Safety Switch
        .6   // Remote Signal Output SW-106 Dumper Safety Switch - Light Curtain
        .7   // Remote Signal Output SW-107 Tank Lid Switch
        .8   // Remote Signal Output DBL-101Tank Level Switch
        .9   // Remote Signal Output Production Cycle Running
   SPARE : DINT;   // Safety Device Output SPARE
   SPARE_IN : DINT := 4;   // Spare Input
        .10   // Drum Dumper Lower Limit Switch N.O.
        .9   // Drum Dumper Upper Limit Switch N.O.
   SPARE_OUT : DINT;
        .0   // SPARE OUTPUT
   ST_S_SW : DINT := 4176;   // Safety Switch Status Output Array
        .0   // Safety Switch Main E-Stop SW104 A/B
        .10   // Light Curtain Obstructed Safety Block Status
        .12   // Saftey Switch Gate SW2 SW108
        .16   // Safety Switch
        .4   // Saftey Switch Gate SW1 SW105
        .6   // Safety Switch Tank Lid Status SW105 A/B
   START_CMPLT : BOOL := 1;   // System Start up Complete
   STARTUP : DINT := 12;   // System Startup Control Bits
   STEAM_ENABLE : ALIAS FOR SIGNAL_OUT_RG_CHOPPER.1;
   STOP_ALL : BOOL;   // Stop All
   STOP_PB_INVERSE : BOOL;   // Inverse of Stop Pushbutton
   SW101_START_PB : BOOL;   // Start PB HMI
   SW102_STOP_PB : BOOL;   // Stop PB HMI
   SW103_CIP_PB : BOOL;   // CIP PB HMI
   SW104_ESTOP : BOOL := 1;   // Safety E-Stop SW-104
   SW105_DEBOUNCE : TIMER := (PRE := 2000, ACC := 2000, EN := 1, DN := 1);   // SW-105 Gate Switch Debounce Timer
   SW105_GATE_SWITCH : BOOL;   // Safety Switch Gate SW #1 SW105 A/B
   SW106_LC : LIGHT_CURTAIN := (ChannelA := 1, ChannelB := 1, InputFilterTime := 10, O1 := 1);   // Safety SW106 Light Curain
   SW106_LIGHT_CUR : BOOL;   // Safety Light Curtain SW-106
   SW107_TANK_LID : BOOL;   // Tank Lid Safety Switch Active
   SW108_DEBOUNCE : TIMER := (PRE := 2000, ACC := 2000, EN := 1, DN := 1);   // SW-108 Gate Switch Debounce Timer
   SW108_GATE_SWITCH : BOOL;   // Safety Switch Gate SW #2 SW108 A/B
   SW109 : BOOL := 1;   // Drum Dumper Upper Limit Switch
   SW109B : BOOL;   // Drum Dumper Upper Limit Switch 2nd Contact
   SW110 : BOOL := 1;   // Drum Dumper Lower Limit Switch
   SW110B : BOOL;   // Drum Dumper Lower Limit Switch 2nd Contact
   SYS_OK : BOOL := 1;   // System OK No Fatal Alarms
   SYS_STRT_RUN : BOOL := 1;   // System Start / Run
   Tank_Lid1 : EMERGENCY_STOP;   // Safety Switch Tank Lid Status SW105 A/B
   TCV101_AM : PUSH_PUSH_PB;   // TCV-101 Temperature Control Man / Auto Push-Push
   TCV101_AO : DINT;   // TCV-101 Temperature Control Valve Analog Out
   TCV101_Auto : BOOL;   // TCV-101 Temp Control Loop Auto
   TCV101_CTL : PID := (CTL := -2080341504, EN := 1, SWM := 1, INI := 1, DVPA := 1, SP := 105.0, KP := 1.0, KI := 0.0002, MAXS := 4095.0, MAXO := 100.0, UPD := 10.0, PV := 52.34, ERR := 52.66, PVH := 200.0, PVDB := 10.0, MAXI := 4095.0, MAXCV := 100.0, MAXTIE := 4095.0, DATA[0] := -1.2859585, DATA[1] := -20.450306, DATA[2] := 52.34, DATA[3] := 52.66, DATA[4] := 105.0, DATA[5] := 0.024420025, DATA[6] := 1.0, DATA[7] := 160.0, DATA[8] := 1.0, DATA[9] := 0.0002, DATA[11] := 1.0, DATA[12] := 0.0002, DATA[15] := 1.0, DATA[16] := 0.024420025);   // PCV-101 PID Temperature Control
        .CTL.26   // PCV-101 PID Switch to Manual
   TCV101_CTL_ST : DINT := 1;   // TCV-101 Control Status 0= Auto 1= Manual 2= Error
   TCV101_Man : BOOL := 1;   // TCV-101 Temp Control Loop Manual
   TCV101_PB : BOOL;   // TCV-101 Temperature Control Man / Auto PB
   TCV101_SP_MAX : REAL := 190.0;   // TCV101 PID Max Temp SP
   TCV101_SP_MIN : REAL := 100.0;   // PCV-101 PID Temp SP MIN
   TEMP1 : BOOL;
   TESTBIT : DINT;   // TEST BIT WORD
   TP3232_TMP_1_Scaled : REAL := 52.34;   // Hot Water Temperature Scaled
   TP3232_TMP_2_Scaled : REAL := 48.38;   // Product Temperature Scaled
   UP_MKBK : BOOL;   // Elevator Down Make / Break LS_U1 Detection
   UP_MKBK1 : BOOL;   // Elevator Up Make / Break Memory 1
   UP_OT_AL : BOOL;   // New Dumper UP Over Travel Alarm
   UP_STP : BOOL;   // Elevator Up STOP
   USER_ON : BOOL;   // There IS a valid HMI User Logged On
   VALV_OUT : REAL;   // TCV-101 Temp Control Valve Pos Output
   WTR_HI_TEMP : BOOL;   // High Water Temperature Alarm
   WTR_HI_TMR : TIMER := (PRE := 10000);   // High Water Temperature Alarm Debounce Timer
END_VAR

PROGRAM FLASH   (* main routine FLASH_1_SEC *)

ROUTINE FLASH_1_SEC   (* ladder *)
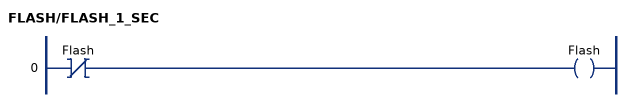
   0: XIO(Flash)OTE(Flash);
END_ROUTINE
END_PROGRAM
